Staubli VAL3: sad_project_1.pjx

--- sad_project_1.pjx ---
Parameters version=s7.7.1 stackSize=5000 millimeterUnit=true
Program file=check_cmt.pgx
Program file=init_prgm.pgx
Program file=launch_print.pgx
Program file=motion_cntl.pgx
Program file=open_socket.pgx
Program file=read_data.pgx
Program file=send_data.pgx
Program file=show_data.pgx
Program file=start.pgx
Program file=stop.pgx
Program file=stop_print.pgx
Data file=sad_project_1.dtx

--- sad_project_1.dtx ---
public num Ref_Vel
public mdesc mNomSpeed = {tmax=100, rmax=100, leave=0.1, reach=0.1, blend=off}
public jointRx Jnt_cnfg = {j3=90, j5=90, j6=90}
public tool tTool = {z=600, rz=55, fatherId=flange[0], ioLink=valve1}
public frame fReference = {x=1365.054, y=-125.975, z=-1150, fatherId=world[0]}
public pointRx Pnt_1st_lyr[2]
  [0] = {y=-1000, rx=-180, rz=-90, shoulder=lefty, elbow=epositive, wrist=wpositive, fatherId=fReference[0]}
  [1] = {y=1000, rx=-180, rz=-90, shoulder=lefty, elbow=epositive, wrist=wpositive, fatherId=fReference[0]}
public pointRx Pnt_2nd_lyr[4]
  [0] = {y=1000, z=77, rx=180, rz=-90, shoulder=lefty, elbow=epositive, wrist=wpositive, fatherId=fReference[0]}
  [1] = {y=-1000, z=77, rx=180, rz=-90, shoulder=lefty, elbow=epositive, wrist=wpositive, fatherId=fReference[0]}
  [2] = {y=-1000, z=22, rx=180, rz=-90, shoulder=lefty, elbow=epositive, wrist=wpositive, fatherId=fReference[0]}
  [3] = {y=1000, z=22, rx=180, rz=-90, shoulder=lefty, elbow=epositive, wrist=wpositive, fatherId=fReference[0]}
public pointRx Pnt_3rd_lyr[4]
  [0] = {y=1000, z=99, rx=180, rz=-90, shoulder=lefty, elbow=epositive, wrist=wpositive, fatherId=fReference[0]}
  [1] = {y=-1000, z=99, rx=180, rz=-90, shoulder=lefty, elbow=epositive, wrist=wpositive, fatherId=fReference[0]}
  [2] = {y=-1000, z=44, rx=180, rz=-90, shoulder=lefty, elbow=epositive, wrist=wpositive, fatherId=fReference[0]}
  [3] = {y=1000, z=44, rx=180, rz=-90, shoulder=lefty, elbow=epositive, wrist=wpositive, fatherId=fReference[0]}
public pointRx Pnt_4th_lyr[4]
  [0] = {y=1000, z=116, rx=180, rz=-90, shoulder=lefty, elbow=epositive, wrist=wpositive, fatherId=fReference[0]}
  [1] = {y=-1000, z=116, rx=180, rz=-90, shoulder=lefty, elbow=epositive, wrist=wpositive, fatherId=fReference[0]}
  [2] = {y=-1000, z=66, rx=180, rz=-90, shoulder=lefty, elbow=epositive, wrist=wpositive, fatherId=fReference[0]}
  [3] = {y=1000, z=66, rx=180, rz=-90, shoulder=lefty, elbow=epositive, wrist=wpositive, fatherId=fReference[0]}
public trsf trTrsf
sio sioASCII = {link=Socket\trsf_sv}
public bool check_status
public bool spd_cntl
public mdesc cnst_vel = {tmax=100, rmax=100, leave=0.1, reach=0.1, blend=cartesian}
aio Tpompe = {link=CanIO\RemIO\remio0_QW}
dio doValve1 = {link=valve1}
dio doValve2 = {link=valve2}
dio doPompe = {link=CanIO\RemIO\remio0_Q}

--- start.pgx ---
program start()
begin
  disablePower()
  cls()
  userPage()
  title(" Concrete 3D Printer-Linear Path ")
  putln("Written by Erfan.")
  setProfile("Manual","123")
  if getProfile() == "Manual"
    putln("Profile is set to Remote Control.")
  endIf
  delay(3)
  enablePower()
  if(watch(isPowered(),3) == false)
    putln("Arm power supply cannot be swithced on.")
  endIf
  putln("Arm power is now switched on.")
  delay(3)
  taskCreate "Initialization",1,init_prgm()
  putln("Pump has been launched.")
  putln("Nozzle is closed.")
  delay(2)
  //taskCreate "SocketOpening",10,open_socket()
  //taskCreate "CheckComnunic",20,check_cmt()
  //wait(check_status == true)
  //delay(2)
  //taskCreate "DataReading",40,read_data()
  //taskCreate "MotionControl",40,motion_cntl()
  //taskCreate "DataDisplay",40,show_data()
  //taskCreate "DataSending",50,send_data()


  //////////////////////////////////////////
  // Go to configuration
  spd_cntl = false
  resetMotion()
  setMonitorSpeed(10)
  movej(Jnt_cnfg[0],tTool[0],cnst_vel[0])
  waitEndMove()

  // Go to Start point - 1st Layer
  spd_cntl = false
  setMonitorSpeed(10)
  movel(Pnt_1st_lyr[0],tTool[0],mNomSpeed[0])
  waitEndMove()

  //**************************************************

  // Printing - 1st Layer
  setProfile("Automatic","123")
  spd_cntl = true
  resetMotion()

  // Starting printing
  call launch_print()

  movel(Pnt_1st_lyr[1],tTool[0],mNomSpeed[0])
  waitEndMove()

  // Stop Printing
  call stop_print()


  //************************************************

  // Go to Start point - 2nd Layer
  resetMotion()
  setProfile("Manual","123")
  spd_cntl = false
  resetMotion()
  setMonitorSpeed(100)
  movel(Pnt_2nd_lyr[0],tTool[0],cnst_vel[0])
  waitEndMove()
  movel(Pnt_2nd_lyr[1],tTool[0],cnst_vel[0])
  waitEndMove()
  movel(Pnt_2nd_lyr[2],tTool[0],cnst_vel[0])
  waitEndMove()

  // Printing - 2nd Layer
  setProfile("Automatic","123")
  spd_cntl = true
  resetMotion()

  // Starting printing
  call launch_print()

  movel(Pnt_2nd_lyr[3],tTool[0],mNomSpeed[0])
  waitEndMove()

  // Stop Printing
  call stop_print()


  //*****************************************

  // Go to Start point - 3rd Layer
  setProfile("Manual","123")
  spd_cntl = false
  resetMotion()
  setMonitorSpeed(100)
  movel(Pnt_3rd_lyr[0],tTool[0],cnst_vel[0])
  waitEndMove()
  movel(Pnt_3rd_lyr[1],tTool[0],cnst_vel[0])
  waitEndMove()
  movel(Pnt_3rd_lyr[2],tTool[0],cnst_vel[0])
  waitEndMove()

  // Printing - 3rd Layer
  setProfile("Automatic","123")
  spd_cntl = true
  resetMotion()

  // Starting printing
  call launch_print()

  movel(Pnt_3rd_lyr[3],tTool[0],mNomSpeed[0])
  waitEndMove()

  // Stop Printing
  call stop_print()

  // **************************************

  // Go to Start point - 4th Layer
  setProfile("Manual","123")
  spd_cntl = false
  resetMotion()
  setMonitorSpeed(100)
  movel(Pnt_4th_lyr[0],tTool[0],cnst_vel[0])
  waitEndMove()
  movel(Pnt_4th_lyr[1],tTool[0],cnst_vel[0])
  waitEndMove()
  movel(Pnt_4th_lyr[2],tTool[0],cnst_vel[0])
  waitEndMove()


  // Printing - 4th Layer
  setProfile("Automatic","123")
  spd_cntl = true
  resetMotion()

  // Printing starts
  call launch_print()

  movel(Pnt_4th_lyr[3],tTool[0],mNomSpeed[0])
  waitEndMove()

  // Stop Printing
  call stop_print()

  // **************************************

  ///////////////////////////
  cls()
  userPage()
  title(" Concrete 3D Printer-Linear Path ")
  putln("printing procedure has been finished.")

  // Go to configuration
  setProfile("Manual","123")
  spd_cntl = false
  resetMotion()
  setMonitorSpeed(100)
  movej(Jnt_cnfg[0],tTool[0],cnst_vel[0])
  waitEndMove()


  /////////////////////

  stopMove()
  disablePower()


  ///////////////////////////////////////////


end

--- open_socket.pgx ---
public program open_socket()
begin

  sioCtrl(sioASCII,"port",11002)
  //sioCtrl(sioASCII,"port",1002)
  //sioCtrl(sioASCII,"target","10.3.1.185")
  //sioCtrl(sioASCII,"target","10.10.5.1")
  sioCtrl(sioASCII,"target","169.254.209.1")
  sioCtrl(sioASCII,"timeout",10)
  sioCtrl(sioASCII,"endOfString",13)
  sioCtrl(sioASCII,"nangle",true)

  putln(" " )
  putln("The communication socket is open.")

  check_status = false

end

--- read_data.pgx ---
public program read_data()
  local string sInputData_1
  local num nRec
  local num nReceived
  local num nInputData_1
begin

  putln("Start to read data !")

  do
    sInputData_1 = ""
    do
      nReceived=sioGet(sioASCII,nRec)
      sInputData_1 = sInputData_1 + chr(nRec)

    until nRec == 13 or nReceived == -1

    if nReceived != 1
      check_status = false
      stopMove()
      cls()
      putln("Communication error !")
      disablePower()
    endIf

    toNum(sInputData_1 , nInputData_1, check_status)

    //put("Reference Velocity [mm/s]: ")
    //put(nInputData_1)
    //putln("")



    if getMoveId() >= 0.05
      Ref_Vel = nInputData_1
    elseIf getMoveId() < 0.05
       Ref_Vel = print_vel
    endIf

   // putln(Ref_Vel)


   delay(0.001)

  until check_status != true

end

--- stop_print.pgx ---
public program stop_print()
begin

      // arrêt pompe
    dioSet(doPompe,0)
    put("Pompe arret")
    // fermeture obturateur
    dioSet(doValve2,0)
    dioSet(doValve1,1)
    put("Obturateur fermé")

end
